PROGRAM GL4_Accumulation
VAR
	GL4: sConveyor;
	GL5: sConveyor;
	RUN_FWD_TO_GL5A_BIT : BOOL; // GL5 EMPTY SO SEND PART FROM GL4 TO GL5
	RUN_FWD_TO_EXIT_BIT : BOOL; // RUN GL4 FWD TO EXIT SENSOR
	GL5A_ENTRY_FTRIG:  F_TRIG;
	
	TEST: BOOL;
END_VAR
VAR // added by the converter: edge detectors and wires of the graphical bodies
    _w1 : BOOL;
END_VAR

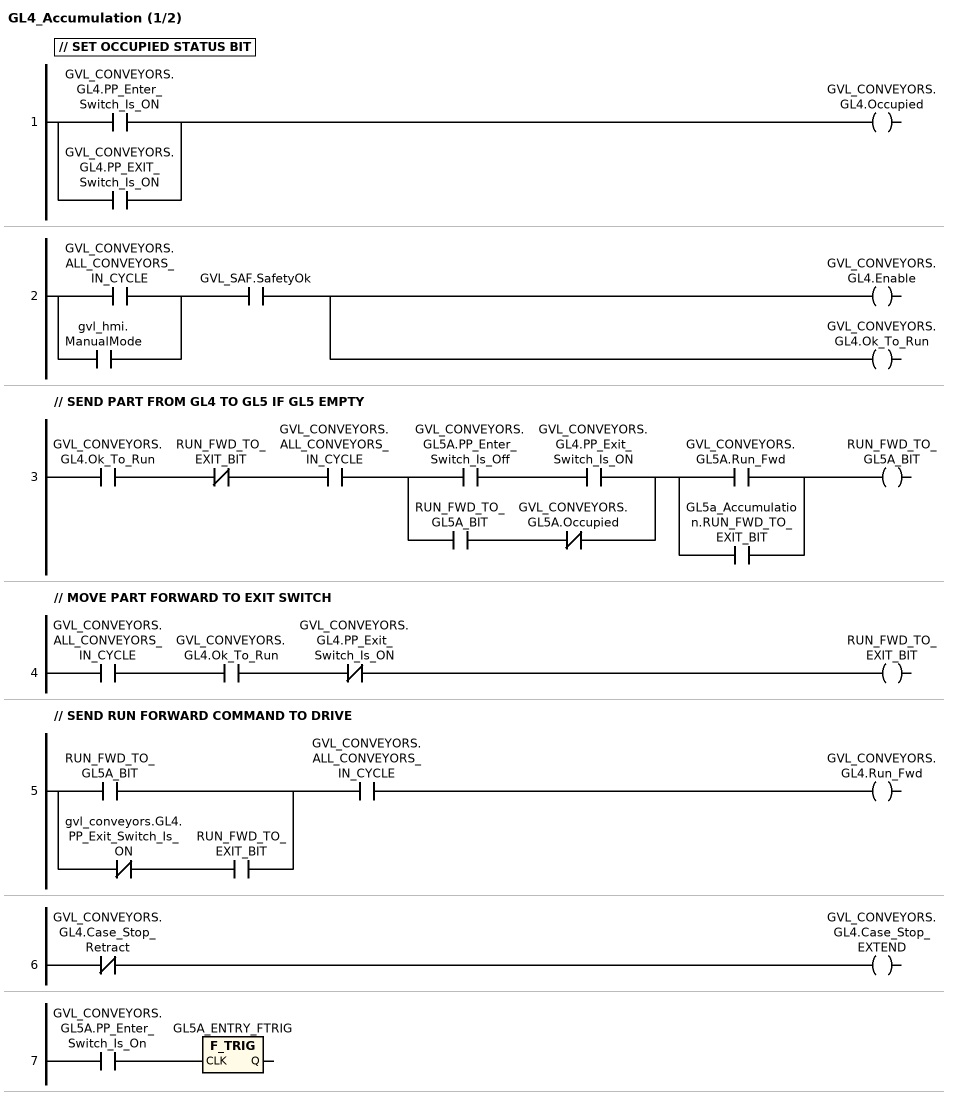
// NETWORK 1
// label: // SET OCCUPIED STATUS BIT
GVL_CONVEYORS.GL4.Occupied := GVL_CONVEYORS.GL4.PP_Enter_Switch_Is_ON OR GVL_CONVEYORS.GL4.PP_EXIT_Switch_Is_ON;

// NETWORK 2
_w1 := (GVL_CONVEYORS.ALL_CONVEYORS_IN_CYCLE OR gvl_hmi.ManualMode) AND GVL_SAF.SafetyOk;
GVL_CONVEYORS.GL4.Enable := _w1;
GVL_CONVEYORS.GL4.Ok_To_Run := _w1;

// NETWORK 3: // SEND PART FROM GL4 TO GL5 IF GL5 EMPTY
RUN_FWD_TO_GL5A_BIT := GVL_CONVEYORS.GL4.Ok_To_Run AND NOT RUN_FWD_TO_EXIT_BIT AND GVL_CONVEYORS.ALL_CONVEYORS_IN_CYCLE AND (GVL_CONVEYORS.GL5A.PP_Enter_Switch_Is_Off AND GVL_CONVEYORS.GL4.PP_Exit_Switch_Is_ON OR RUN_FWD_TO_GL5A_BIT AND NOT GVL_CONVEYORS.GL5A.Occupied) AND (GVL_CONVEYORS.GL5A.Run_Fwd OR GL5a_Accumulation.RUN_FWD_TO_EXIT_BIT);

// NETWORK 4: // MOVE PART FORWARD TO EXIT SWITCH
RUN_FWD_TO_EXIT_BIT := GVL_CONVEYORS.ALL_CONVEYORS_IN_CYCLE AND GVL_CONVEYORS.GL4.Ok_To_Run AND NOT GVL_CONVEYORS.GL4.PP_Exit_Switch_Is_ON;

// NETWORK 5: // SEND RUN FORWARD COMMAND TO DRIVE
GVL_CONVEYORS.GL4.Run_Fwd := (RUN_FWD_TO_GL5A_BIT OR NOT gvl_conveyors.GL4.PP_Exit_Switch_Is_ON AND RUN_FWD_TO_EXIT_BIT) AND GVL_CONVEYORS.ALL_CONVEYORS_IN_CYCLE;

// NETWORK 6
GVL_CONVEYORS.GL4.Case_Stop_EXTEND := NOT GVL_CONVEYORS.GL4.Case_Stop_Retract;

// NETWORK 7
GL5A_ENTRY_FTRIG(CLK := GVL_CONVEYORS.GL5A.PP_Enter_Switch_Is_On); // F_TRIG

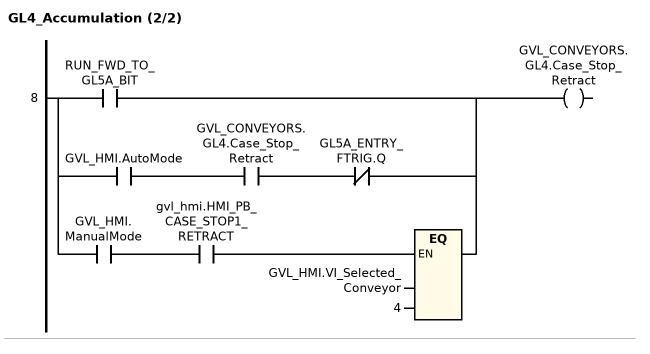
// NETWORK 8
GVL_CONVEYORS.GL4.Case_Stop_Retract := RUN_FWD_TO_GL5A_BIT OR GVL_HMI.AutoMode AND GVL_CONVEYORS.GL4.Case_Stop_Retract AND NOT GL5A_ENTRY_FTRIG.Q OR GVL_HMI.ManualMode AND gvl_hmi.HMI_PB_CASE_STOP1_RETRACT AND GVL_HMI.VI_Selected_Conveyor = 4;

END_PROGRAM

(* stored: Version 1.1.0.1, ProductVersion 3.1.4024.12
   POU GL4_Accumulation: Id {dad9f2aa-0fa0-4f46-be24-203a42a4bdd4}, SpecialFunc None *)
